SUBAPPLICATION Uebung_020j2_AX (* DigitalInput_I1 auf DigitalOutput_Q1/2; 2xAX_TP; Impulsformend mit SUB *)
  (* Standard: 61499-2; Description: Copyright (c) 2023 Meisterschulen am Ostbahnhof This program and the accompanying materials are made available under the terms of the Eclipse Public License 2.0 which is available at https://www.eclipse.org/legal/epl-2.0/ SPDX-License-Identifier: EPL-2.0 *)
  (* Version 1.0, 2026-01-16, Franz Höpfinger, Meisterschulen am Ostbahnhof, initial API and implementation and/or initial documentation *)
  PACKAGE Uebungen;
  IMPORT logiBUS::io::DI::logiBUS_DI::Input_I1;
  IMPORT logiBUS::io::DQ::logiBUS_DO::Output_Q1;
  IMPORT logiBUS::io::DQ::logiBUS_DO::Output_Q2;
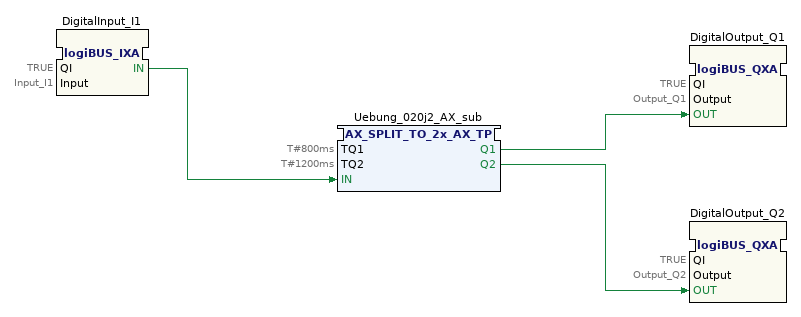
  FBS
    DigitalInput_I1 : logiBUS::io::DI::logiBUS_IXA(QI := TRUE, Input := Input_I1);
    DigitalOutput_Q1 : logiBUS::io::DQ::logiBUS_QXA(QI := TRUE, Output := Output_Q1);
    DigitalOutput_Q2 : logiBUS::io::DQ::logiBUS_QXA(QI := TRUE, Output := Output_Q2);
  END_FBS
  SUBAPPS
    Uebung_020j2_AX_sub : MyLib::sys::AX_SPLIT_TO_2x_AX_TP(TQ1 := T#800ms, TQ2 := T#1200ms);
  END_SUBAPPS
  ADAPTER_CONNECTIONS
    DigitalInput_I1.IN TO Uebung_020j2_AX_sub.IN;
    Uebung_020j2_AX_sub.Q1 TO DigitalOutput_Q1.OUT;
    Uebung_020j2_AX_sub.Q2 TO DigitalOutput_Q2.OUT;
  END_CONNECTIONS
END_SUBAPPLICATION
